TYPE ST_motion :
STRUCT
	bEnable   : BOOL;
    bStop     : BOOL;
    bMoveRel  : BOOL;
    rVelocity : REAL;
    rDistance : REAL;
END_STRUCT
END_TYPE

(* stored: Version 1.1.0.1, ProductVersion 3.1.4026.18
   DUT ST_motion: Id {3f38c839-4db6-4531-84a6-199bc4689f56} *)
